% RSLogix 500 project TESTE 1100 WT21-CS MODBUS WT.RSS, saved by version 11.00.00.00 %
PROJECT "UNTITLED"    % processor: Bul.1763 MicroLogix 1100 Series A %

PROGRAM FILES
  LAD 2   5 rungs

DATA FILES
  O0 OUTPUT  4 elements
  I1 INPUT  6 elements
  S2 STATUS  66 elements
  B3 BINARY  1 elements
  T4 TIMER  1 elements
  C5 COUNTER  1 elements
  R6 CONTROL  1 elements
  N7 INTEGER  10 elements
  F8 FLOAT  2 elements
  L9 PESOS  10 elements
  MG11 MODBUS  3 elements

LADDER 2
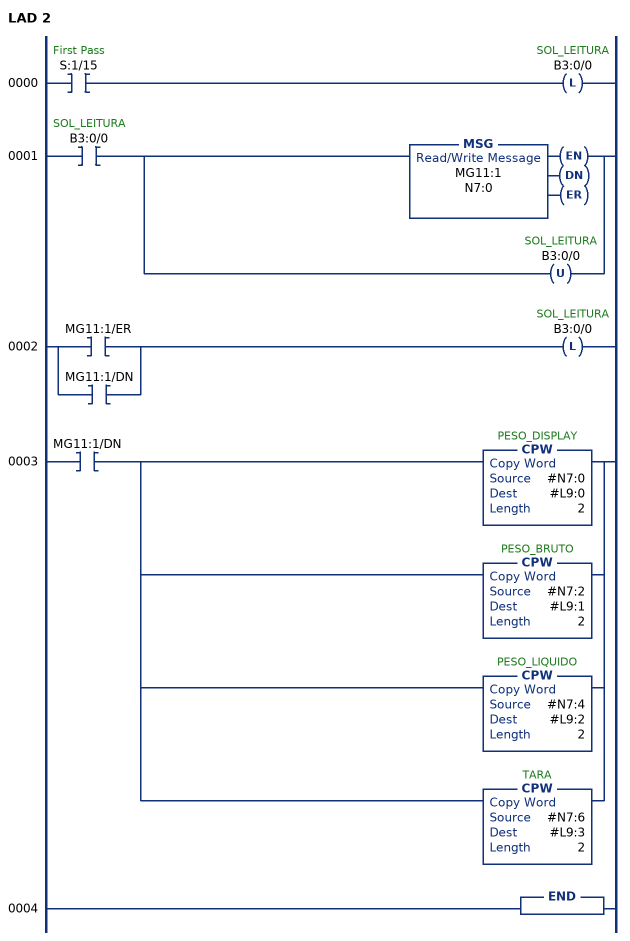
% Rung: 0 %
SOR XIC S:1/15 OTL B3:0/0 EOR
%   S:1/15  "First Pass" %
%   B3:0/0  SOL_LEITURA %
% Rung: 1 %
SOR XIC B3:0/0 BST MSG MG11:1 N7:0 NXB OTU B3:0/0 BND EOR
%   B3:0/0  SOL_LEITURA %
%   MSG set-up: 03 Read Holding Registers (4xxxxx) | 3 | 8 | 1 | N7:0 | 0 | 9 | 0 | CLIENT | 0 | 0 | ? %
% Rung: 2 %
SOR BST XIC MG11:1/ER NXB XIC MG11:1/DN BND OTL B3:0/0 EOR
%   B3:0/0  SOL_LEITURA %
% Rung: 3 %
SOR XIC MG11:1/DN BST CPW #N7:0 #L9:0 2 NXB CPW #N7:2 #L9:1 2 NXB CPW #N7:4 #L9:2 2 NXB CPW #N7:6 #L9:3 2 BND EOR
%   L9:0  PESO_DISPLAY %
%   L9:1  PESO_BRUTO %
%   L9:2  PESO_LIQUIDO %
%   L9:3  TARA %
% Rung: 4 %
SOR END EOR

DATA TABLE (non-zero values as saved)
DATA B3
% B3:0 % 0X0060
DATA N7
% N7:0 % 0 0 -2 -1 0 0 -2 -1 0 0
DATA F8
% F8:0 % nan 0
DATA L9
% L9:0 % 0 -2 0 -2 0
